Omron CX-Programmer project 新工程 (CX-Programmer 9.60)

# PLC 新PLC1: CP1L-E EL

## Global symbols (name address type ; comment)
10 CHANNEL  ; 10
T0001 BOOL  ; DT1定时器

## Program 新程序1 (cyclic task 0)

### Section 段1

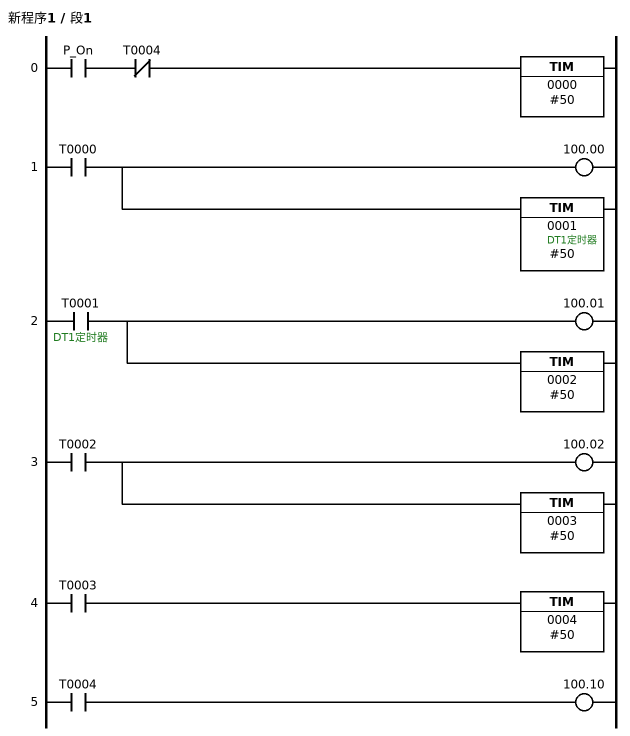
; rung 0
LD P_On
ANDNOT T0004
TIM 0000 #50
; rung 1
LD T0000
OUT 100.00
TIM 0001 #50  ; DT1定时器
; rung 2
LD T0001  ; DT1定时器
OUT 100.01
TIM 0002 #50
; rung 3
LD T0002
OUT 100.02
TIM 0003 #50
; rung 4
LD T0003
TIM 0004 #50
; rung 5
LD T0004
OUT 100.10

### Section END
; rung 0
END(001)